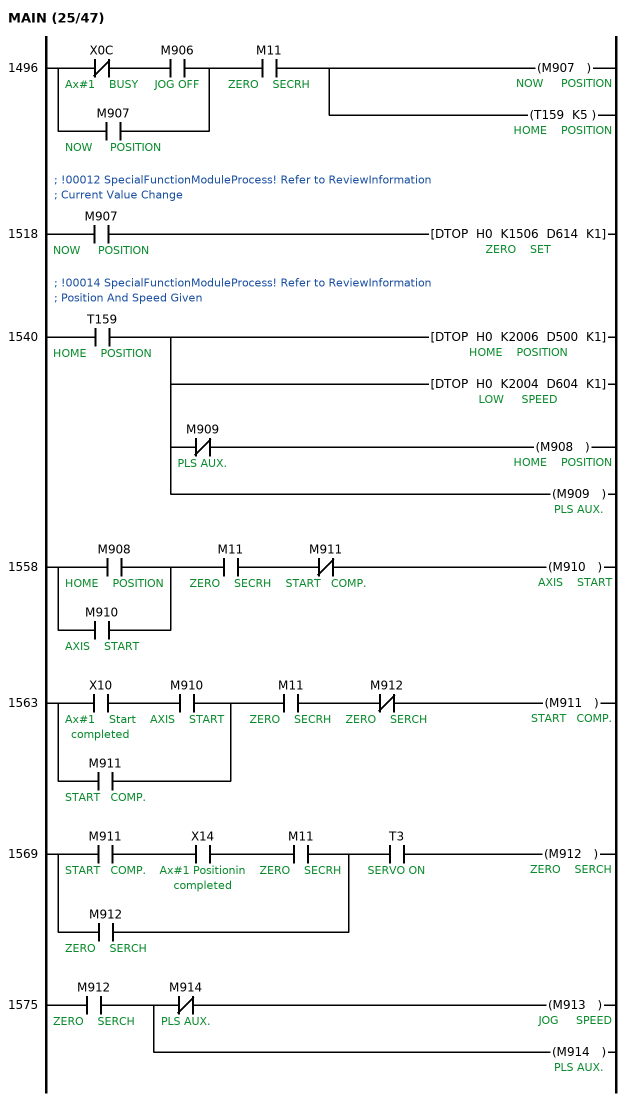
[picture p24: ladder of MAIN, rungs at steps 1496 to 1575]
1496  LDI     X0C  ; Ax#1    BUSY
      AND     M906  ; JOG OFF
      OR      M907  ; NOW     POSITION
      AND     M11  ; ZERO    SECRH
      OUT     M907  ; NOW     POSITION
      OUT     T159 K5  ; HOME    POSITION
; !00012 SpecialFunctionModuleProcess! Refer to ReviewInformation
; Current Value Change
1518  LD      M907  ; NOW     POSITION
      DTOP    H0 K1506 D614 K1
; !00014 SpecialFunctionModuleProcess! Refer to ReviewInformation
; Position And Speed Given
1540  LD      T159  ; HOME    POSITION
      DTOP    H0 K2006 D500 K1
      DTOP    H0 K2004 D604 K1
      MPS
      ANI     M909  ; PLS AUX.
      OUT     M908  ; HOME    POSITION
      MPP
      OUT     M909  ; PLS AUX.
1558  LD      M908  ; HOME    POSITION
      OR      M910  ; AXIS    START
      AND     M11  ; ZERO    SECRH
      ANI     M911  ; START   COMP.
      OUT     M910  ; AXIS    START
1563  LD      X10  ; Ax#1    Start   completed
      AND     M910  ; AXIS    START
      OR      M911  ; START   COMP.
      AND     M11  ; ZERO    SECRH
      ANI     M912  ; ZERO    SERCH
      OUT     M911  ; START   COMP.
1569  LD      M911  ; START   COMP.
      AND     X14  ; Ax#1 Positionin completed
      AND     M11  ; ZERO    SECRH
      OR      M912  ; ZERO    SERCH
      AND     T3  ; SERVO ON
      OUT     M912  ; ZERO    SERCH
1575  LD      M912  ; ZERO    SERCH
      MPS
      ANI     M914  ; PLS AUX.
      OUT     M913  ; JOG     SPEED
      MPP
      OUT     M914  ; PLS AUX.
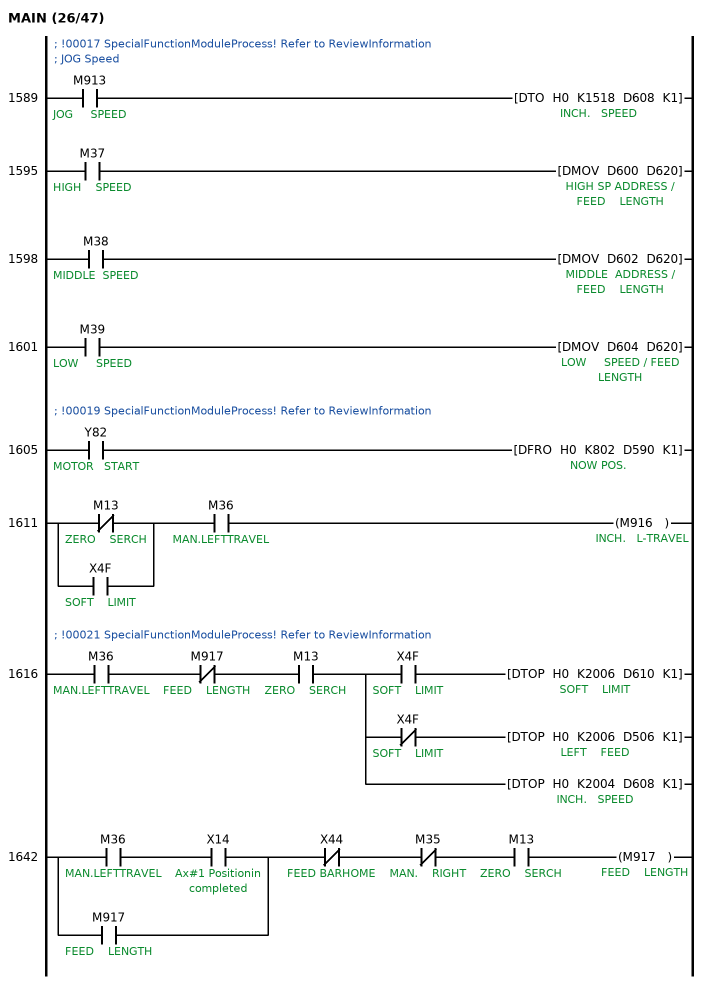
; !00017 SpecialFunctionModuleProcess! Refer to ReviewInformation
; JOG Speed
1589  LD      M913  ; JOG     SPEED
      DTO     H0 K1518 D608 K1
1595  LD      M37  ; HIGH    SPEED
      DMOV    D600 D620  ; FEED    LENGTH
1598  LD      M38  ; MIDDLE  SPEED
      DMOV    D602 D620
1601  LD      M39  ; LOW     SPEED
      DMOV    D604 D620
; !00019 SpecialFunctionModuleProcess! Refer to ReviewInformation
1605  LD      Y82  ; MOTOR   START
      DFRO    H0 K802 D590 K1
1611  LDI     M13  ; ZERO    SERCH
      OR      X4F  ; SOFT    LIMIT
      AND     M36  ; MAN.LEFTTRAVEL
      OUT     M916  ; INCH.   L-TRAVEL
; !00021 SpecialFunctionModuleProcess! Refer to ReviewInformation
1616  LD      M36  ; MAN.LEFTTRAVEL
      ANI     M917  ; FEED    LENGTH
      AND     M13  ; ZERO    SERCH
      MPS
      AND     X4F  ; SOFT    LIMIT
      DTOP    H0 K2006 D610 K1
      MRD
      ANI     X4F  ; SOFT    LIMIT
      DTOP    H0 K2006 D506 K1  ; LEFT    FEED
      MPP
      DTOP    H0 K2004 D608 K1
1642  LD      M36  ; MAN.LEFTTRAVEL
      AND     X14  ; Ax#1 Positionin completed
      OR      M917  ; FEED    LENGTH
      ANI     X44  ; FEED BARHOME
      ANI     M35  ; MAN.    RIGHT
      AND     M13  ; ZERO    SERCH
      OUT     M917  ; FEED    LENGTH
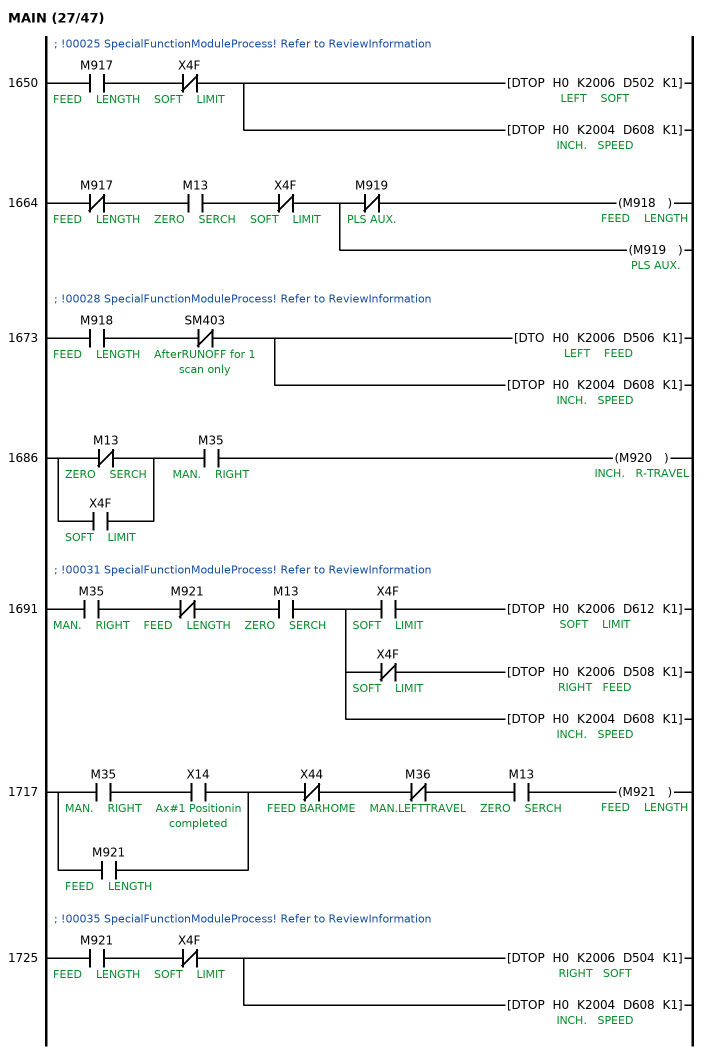
; !00025 SpecialFunctionModuleProcess! Refer to ReviewInformation
1650  LD      M917  ; FEED    LENGTH
      ANI     X4F  ; SOFT    LIMIT
      DTOP    H0 K2006 D502 K1
      DTOP    H0 K2004 D608 K1
1664  LDI     M917  ; FEED    LENGTH
      AND     M13  ; ZERO    SERCH
      ANI     X4F  ; SOFT    LIMIT
      MPS
      ANI     M919  ; PLS AUX.
      OUT     M918  ; FEED    LENGTH
      MPP
      OUT     M919  ; PLS AUX.
; !00028 SpecialFunctionModuleProcess! Refer to ReviewInformation
1673  LD      M918  ; FEED    LENGTH
      ANI     SM403  ; AfterRUNOFF for 1  scan only
      DTO     H0 K2006 D506 K1
      DTOP    H0 K2004 D608 K1
1686  LDI     M13  ; ZERO    SERCH
      OR      X4F  ; SOFT    LIMIT
      AND     M35  ; MAN.    RIGHT
      OUT     M920  ; INCH.   R-TRAVEL
; !00031 SpecialFunctionModuleProcess! Refer to ReviewInformation
1691  LD      M35  ; MAN.    RIGHT
      ANI     M921  ; FEED    LENGTH
      AND     M13  ; ZERO    SERCH
      MPS
      AND     X4F  ; SOFT    LIMIT
      DTOP    H0 K2006 D612 K1
      MRD
      ANI     X4F  ; SOFT    LIMIT
      DTOP    H0 K2006 D508 K1  ; RIGHT   FEED
      MPP
      DTOP    H0 K2004 D608 K1
1717  LD      M35  ; MAN.    RIGHT
      AND     X14  ; Ax#1 Positionin completed
      OR      M921  ; FEED    LENGTH
      ANI     X44  ; FEED BARHOME
      ANI     M36  ; MAN.LEFTTRAVEL
      AND     M13  ; ZERO    SERCH
      OUT     M921  ; FEED    LENGTH
; !00035 SpecialFunctionModuleProcess! Refer to ReviewInformation
1725  LD      M921  ; FEED    LENGTH
      ANI     X4F  ; SOFT    LIMIT
      DTOP    H0 K2006 D504 K1
      DTOP    H0 K2004 D608 K1
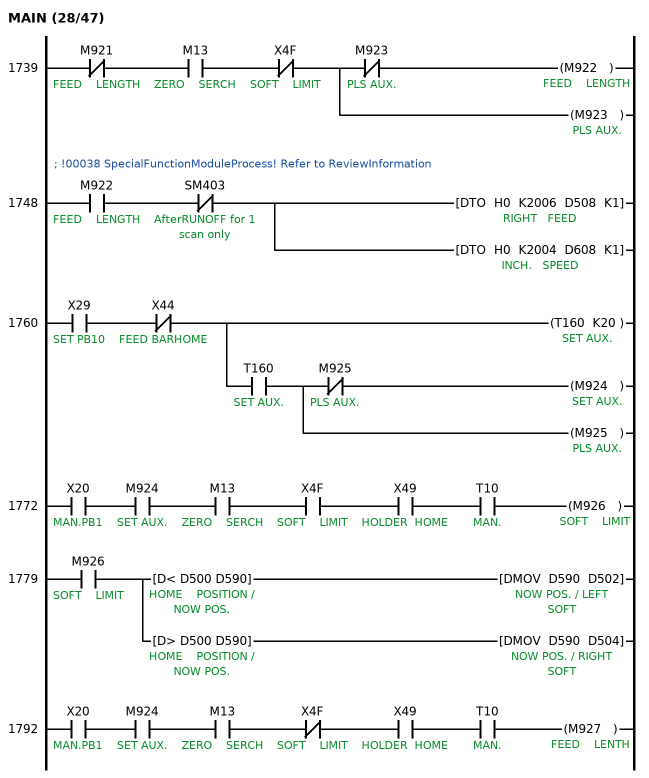
1739  LDI     M921  ; FEED    LENGTH
      AND     M13  ; ZERO    SERCH
      ANI     X4F  ; SOFT    LIMIT
      MPS
      ANI     M923  ; PLS AUX.
      OUT     M922  ; FEED    LENGTH
      MPP
      OUT     M923  ; PLS AUX.
; !00038 SpecialFunctionModuleProcess! Refer to ReviewInformation
1748  LD      M922  ; FEED    LENGTH
      ANI     SM403  ; AfterRUNOFF for 1  scan only
      DTO     H0 K2006 D508 K1
      DTO     H0 K2004 D608 K1
1760  LD      X29  ; SET PB10
      ANI     X44  ; FEED BARHOME
      OUT     T160 K20  ; SET AUX.
      AND     T160  ; SET AUX.
      MPS
      ANI     M925  ; PLS AUX.
      OUT     M924  ; SET AUX.
      MPP
      OUT     M925  ; PLS AUX.
1772  LD      X20  ; MAN.PB1
      AND     M924  ; SET AUX.
      AND     M13  ; ZERO    SERCH
      AND     X4F  ; SOFT    LIMIT
      AND     X49  ; HOLDER  HOME
      AND     T10  ; MAN.
      OUT     M926  ; SOFT    LIMIT
1779  LD      M926  ; SOFT    LIMIT
      MPS
      ANDD<   D500 D590  ; HOME    POSITION / NOW POS.
      DMOV    D590 D502
      MPP
      ANDD>   D500 D590  ; HOME    POSITION / NOW POS.
      DMOV    D590 D504
1792  LD      X20  ; MAN.PB1
      AND     M924  ; SET AUX.
      AND     M13  ; ZERO    SERCH
      ANI     X4F  ; SOFT    LIMIT
      AND     X49  ; HOLDER  HOME
      AND     T10  ; MAN.
      OUT     M927  ; FEED    LENTH
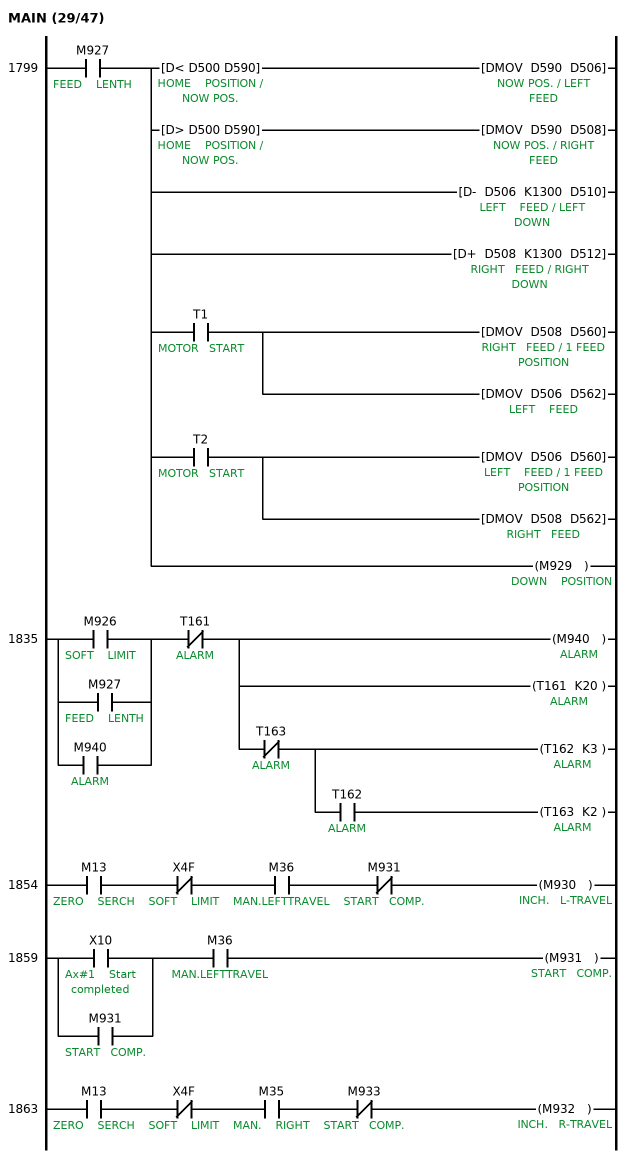
1799  LD      M927  ; FEED    LENTH
      MPS
      ANDD<   D500 D590  ; HOME    POSITION / NOW POS.
      DMOV    D590 D506
      MRD
      ANDD>   D500 D590  ; HOME    POSITION / NOW POS.
      DMOV    D590 D508
      MPP
      D-      D506 K1300 D510  ; LEFT    DOWN
      D+      D508 K1300 D512  ; RIGHT   DOWN
      MPS
      AND     T1  ; MOTOR   START
      DMOV    D508 D560  ; 1 FEED  POSITION
      DMOV    D506 D562
      MRD
      AND     T2  ; MOTOR   START
      DMOV    D506 D560
      DMOV    D508 D562
      MPP
      OUT     M929  ; DOWN    POSITION
1835  LD      M926  ; SOFT    LIMIT
      OR      M927  ; FEED    LENTH
      OR      M940  ; ALARM
      ANI     T161  ; ALARM
      OUT     M940  ; ALARM
      OUT     T161 K20  ; ALARM
      ANI     T163  ; ALARM
      OUT     T162 K3  ; ALARM
      AND     T162  ; ALARM
      OUT     T163 K2  ; ALARM
1854  LD      M13  ; ZERO    SERCH
      ANI     X4F  ; SOFT    LIMIT
      AND     M36  ; MAN.LEFTTRAVEL
      ANI     M931  ; START   COMP.
      OUT     M930  ; INCH.   L-TRAVEL
1859  LD      X10  ; Ax#1    Start   completed
      OR      M931  ; START   COMP.
      AND     M36  ; MAN.LEFTTRAVEL
      OUT     M931  ; START   COMP.
1863  LD      M13  ; ZERO    SERCH
      ANI     X4F  ; SOFT    LIMIT
      AND     M35  ; MAN.    RIGHT
      ANI     M933  ; START   COMP.
      OUT     M932  ; INCH.   R-TRAVEL
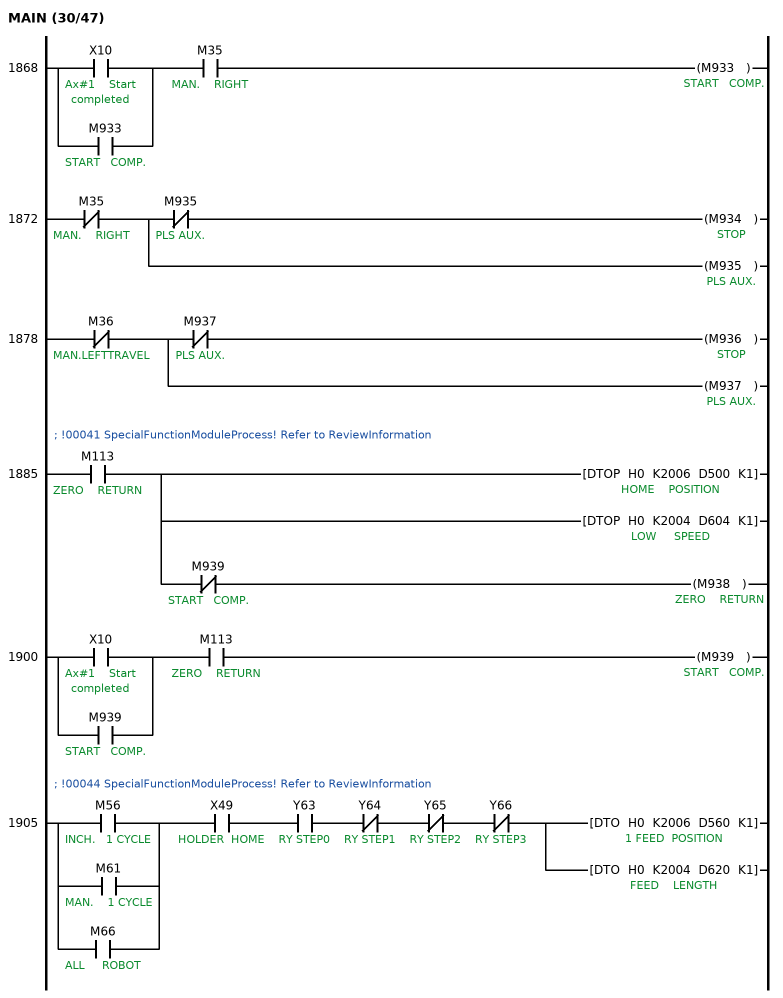
1868  LD      X10  ; Ax#1    Start   completed
      OR      M933  ; START   COMP.
      AND     M35  ; MAN.    RIGHT
      OUT     M933  ; START   COMP.
1872  LDI     M35  ; MAN.    RIGHT
      MPS
      ANI     M935  ; PLS AUX.
      OUT     M934  ; STOP
      MPP
      OUT     M935  ; PLS AUX.
1878  LDI     M36  ; MAN.LEFTTRAVEL
      MPS
      ANI     M937  ; PLS AUX.
      OUT     M936  ; STOP
      MPP
      OUT     M937  ; PLS AUX.
; !00041 SpecialFunctionModuleProcess! Refer to ReviewInformation
1885  LD      M113  ; ZERO    RETURN
      DTOP    H0 K2006 D500 K1
      DTOP    H0 K2004 D604 K1
      ANI     M939  ; START   COMP.
      OUT     M938  ; ZERO    RETURN
1900  LD      X10  ; Ax#1    Start   completed
      OR      M939  ; START   COMP.
      AND     M113  ; ZERO    RETURN
      OUT     M939  ; START   COMP.
; !00044 SpecialFunctionModuleProcess! Refer to ReviewInformation
1905  LD      M56  ; INCH.   1 CYCLE
      OR      M61  ; MAN.    1 CYCLE
      OR      M66  ; ALL     ROBOT
      AND     X49  ; HOLDER  HOME
      AND     Y63  ; RY STEP0
      ANI     Y64  ; RY STEP1
      ANI     Y65  ; RY STEP2
      ANI     Y66  ; RY STEP3
      DTO     H0 K2006 D560 K1
      DTO     H0 K2004 D620 K1
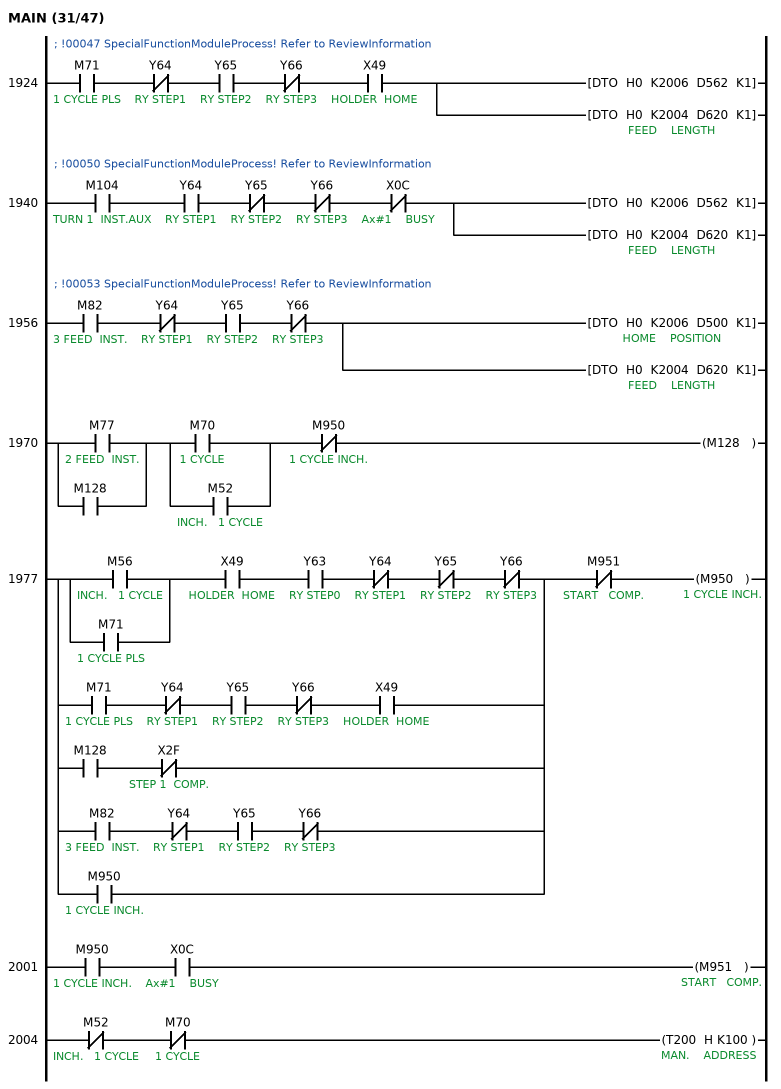
; !00047 SpecialFunctionModuleProcess! Refer to ReviewInformation
1924  LD      M71  ; 1 CYCLE PLS
      ANI     Y64  ; RY STEP1
      AND     Y65  ; RY STEP2
      ANI     Y66  ; RY STEP3
      AND     X49  ; HOLDER  HOME
      DTO     H0 K2006 D562 K1
      DTO     H0 K2004 D620 K1
; !00050 SpecialFunctionModuleProcess! Refer to ReviewInformation
1940  LD      M104  ; TURN 1  INST.AUX
      AND     Y64  ; RY STEP1
      ANI     Y65  ; RY STEP2
      ANI     Y66  ; RY STEP3
      ANI     X0C  ; Ax#1    BUSY
      DTO     H0 K2006 D562 K1
      DTO     H0 K2004 D620 K1
; !00053 SpecialFunctionModuleProcess! Refer to ReviewInformation
1956  LD      M82  ; 3 FEED  INST.
      ANI     Y64  ; RY STEP1
      AND     Y65  ; RY STEP2
      ANI     Y66  ; RY STEP3
      DTO     H0 K2006 D500 K1
      DTO     H0 K2004 D620 K1
1970  LD      M77  ; 2 FEED  INST.
      OR      M128
      LD      M70  ; 1 CYCLE
      OR      M52  ; INCH.   1 CYCLE
      ANB
      ANI     M950  ; 1 CYCLE INCH.
      OUT     M128
1977  LD      M56  ; INCH.   1 CYCLE
      OR      M71  ; 1 CYCLE PLS
      AND     X49  ; HOLDER  HOME
      AND     Y63  ; RY STEP0
      ANI     Y64  ; RY STEP1
      ANI     Y65  ; RY STEP2
      ANI     Y66  ; RY STEP3
      LD      M71  ; 1 CYCLE PLS
      ANI     Y64  ; RY STEP1
      AND     Y65  ; RY STEP2
      ANI     Y66  ; RY STEP3
      AND     X49  ; HOLDER  HOME
      ORB
      LD      M128
      ANI     X2F  ; STEP 1  COMP.
      ORB
      LD      M82  ; 3 FEED  INST.
      ANI     Y64  ; RY STEP1
      AND     Y65  ; RY STEP2
      ANI     Y66  ; RY STEP3
      ORB
      OR      M950  ; 1 CYCLE INCH.
      ANI     M951  ; START   COMP.
      OUT     M950  ; 1 CYCLE INCH.
2001  LD      M950  ; 1 CYCLE INCH.
      AND     X0C  ; Ax#1    BUSY
      OUT     M951  ; START   COMP.
2004  LDI     M52  ; INCH.   1 CYCLE
      ANI     M70  ; 1 CYCLE
      OUTH    T200 K100  ; MAN.    ADDRESS
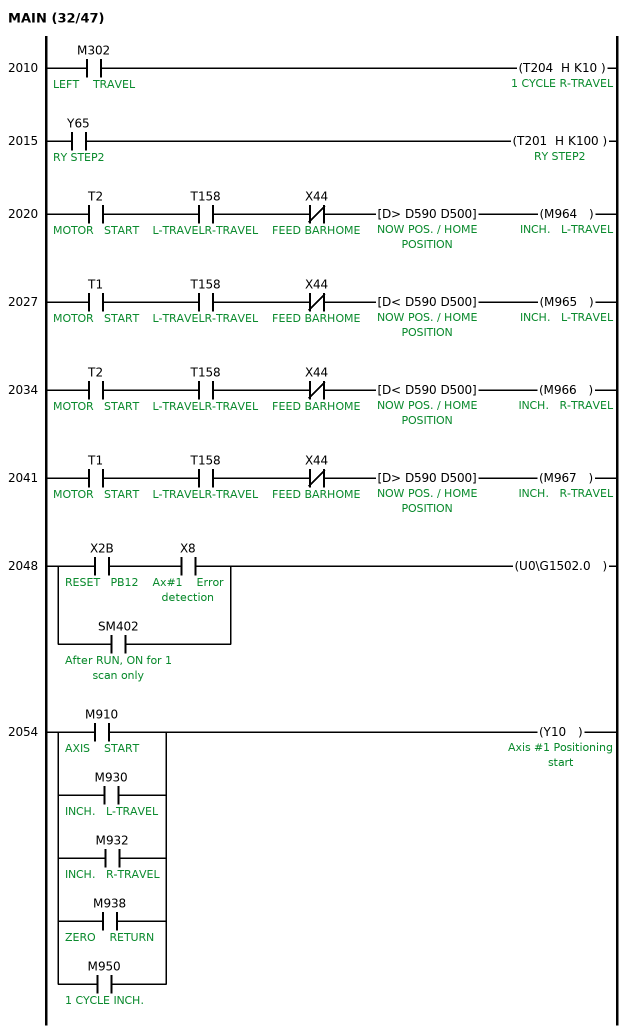
2010  LD      M302  ; LEFT    TRAVEL
      OUTH    T204 K10  ; 1 CYCLE R-TRAVEL
2015  LD      Y65  ; RY STEP2
      OUTH    T201 K100  ; RY STEP2
2020  LD      T2  ; MOTOR   START
      AND     T158  ; L-TRAVELR-TRAVEL
      ANI     X44  ; FEED BARHOME
      ANDD>   D590 D500  ; NOW POS. / HOME    POSITION
      OUT     M964  ; INCH.   L-TRAVEL
2027  LD      T1  ; MOTOR   START
      AND     T158  ; L-TRAVELR-TRAVEL
      ANI     X44  ; FEED BARHOME
      ANDD<   D590 D500  ; NOW POS. / HOME    POSITION
      OUT     M965  ; INCH.   L-TRAVEL
2034  LD      T2  ; MOTOR   START
      AND     T158  ; L-TRAVELR-TRAVEL
      ANI     X44  ; FEED BARHOME
      ANDD<   D590 D500  ; NOW POS. / HOME    POSITION
      OUT     M966  ; INCH.   R-TRAVEL
2041  LD      T1  ; MOTOR   START
      AND     T158  ; L-TRAVELR-TRAVEL
      ANI     X44  ; FEED BARHOME
      ANDD>   D590 D500  ; NOW POS. / HOME    POSITION
      OUT     M967  ; INCH.   R-TRAVEL
2048  LD      X2B  ; RESET   PB12
      AND     X8  ; Ax#1    Error   detection
      OR      SM402  ; After RUN, ON for 1 scan only
      OUT     U0\G1502.0
2054  LD      M910  ; AXIS    START
      OR      M930  ; INCH.   L-TRAVEL
      OR      M932  ; INCH.   R-TRAVEL
      OR      M938  ; ZERO    RETURN
      OR      M950  ; 1 CYCLE INCH.
      OUT     Y10  ; Axis #1 Positioning start
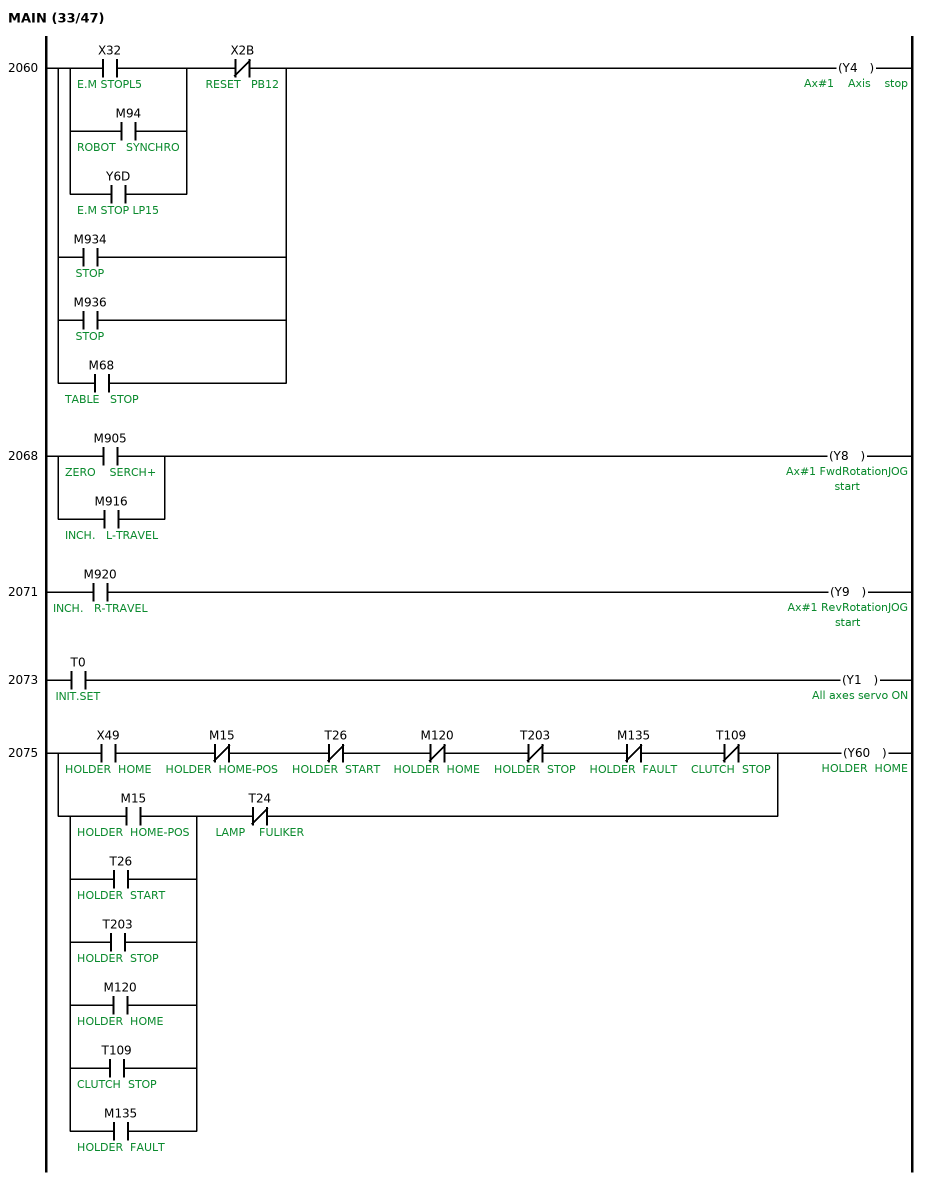
2060  LD      X32  ; E.M STOPL5
      OR      M94  ; ROBOT   SYNCHRO
      OR      Y6D  ; E.M STOP LP15
      ANI     X2B  ; RESET   PB12
      OR      M934  ; STOP
      OR      M936  ; STOP
      OR      M68  ; TABLE   STOP
      OUT     Y4  ; Ax#1    Axis    stop
2068  LD      M905  ; ZERO    SERCH+
      OR      M916  ; INCH.   L-TRAVEL
      OUT     Y8  ; Ax#1 FwdRotationJOG     start
2071  LD      M920  ; INCH.   R-TRAVEL
      OUT     Y9  ; Ax#1 RevRotationJOG     start
2073  LD      T0  ; INIT.SET
      OUT     Y1  ; All axes servo ON
2075  LD      X49  ; HOLDER  HOME
      ANI     M15  ; HOLDER  HOME-POS
      ANI     T26  ; HOLDER  START
      ANI     M120  ; HOLDER  HOME
      ANI     T203  ; HOLDER  STOP
      ANI     M135  ; HOLDER  FAULT
      ANI     T109  ; CLUTCH  STOP
      LD      M15  ; HOLDER  HOME-POS
      OR      T26  ; HOLDER  START
      OR      T203  ; HOLDER  STOP
      OR      M120  ; HOLDER  HOME
      OR      T109  ; CLUTCH  STOP
      OR      M135  ; HOLDER  FAULT
      ANI     T24  ; LAMP    FULIKER
      ORB
      OUT     Y60  ; HOLDER  HOME
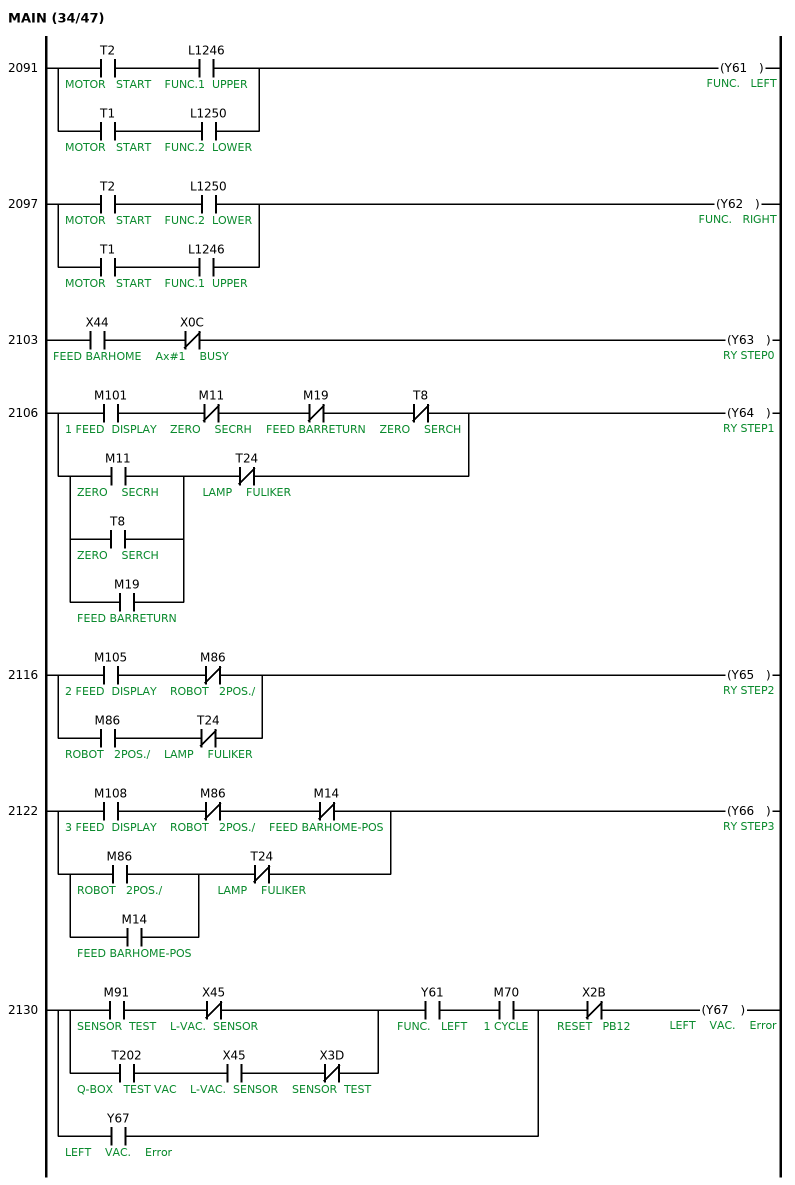
2091  LD      T2  ; MOTOR   START
      AND     L1246  ; FUNC.1  UPPER
      LD      T1  ; MOTOR   START
      AND     L1250  ; FUNC.2  LOWER
      ORB
      OUT     Y61  ; FUNC.   LEFT
2097  LD      T2  ; MOTOR   START
      AND     L1250  ; FUNC.2  LOWER
      LD      T1  ; MOTOR   START
      AND     L1246  ; FUNC.1  UPPER
      ORB
      OUT     Y62  ; FUNC.   RIGHT
2103  LD      X44  ; FEED BARHOME
      ANI     X0C  ; Ax#1    BUSY
      OUT     Y63  ; RY STEP0
2106  LD      M101  ; 1 FEED  DISPLAY
      ANI     M11  ; ZERO    SECRH
      ANI     M19  ; FEED BARRETURN
      ANI     T8  ; ZERO    SERCH
      LD      M11  ; ZERO    SECRH
      OR      T8  ; ZERO    SERCH
      OR      M19  ; FEED BARRETURN
      ANI     T24  ; LAMP    FULIKER
      ORB
      OUT     Y64  ; RY STEP1
2116  LD      M105  ; 2 FEED  DISPLAY
      ANI     M86  ; ROBOT   2POS./
      LD      M86  ; ROBOT   2POS./
      ANI     T24  ; LAMP    FULIKER
      ORB
      OUT     Y65  ; RY STEP2
2122  LD      M108  ; 3 FEED  DISPLAY
      ANI     M86  ; ROBOT   2POS./
      ANI     M14  ; FEED BARHOME-POS
      LD      M86  ; ROBOT   2POS./
      OR      M14  ; FEED BARHOME-POS
      ANI     T24  ; LAMP    FULIKER
      ORB
      OUT     Y66  ; RY STEP3
2130  LD      M91  ; SENSOR  TEST
      ANI     X45  ; L-VAC.  SENSOR
      LD      T202  ; Q-BOX   TEST VAC
      AND     X45  ; L-VAC.  SENSOR
      ANI     X3D  ; SENSOR  TEST
      ORB
      AND     Y61  ; FUNC.   LEFT
      AND     M70  ; 1 CYCLE
      OR      Y67  ; LEFT    VAC.    Error
      ANI     X2B  ; RESET   PB12
      OUT     Y67  ; LEFT    VAC.    Error
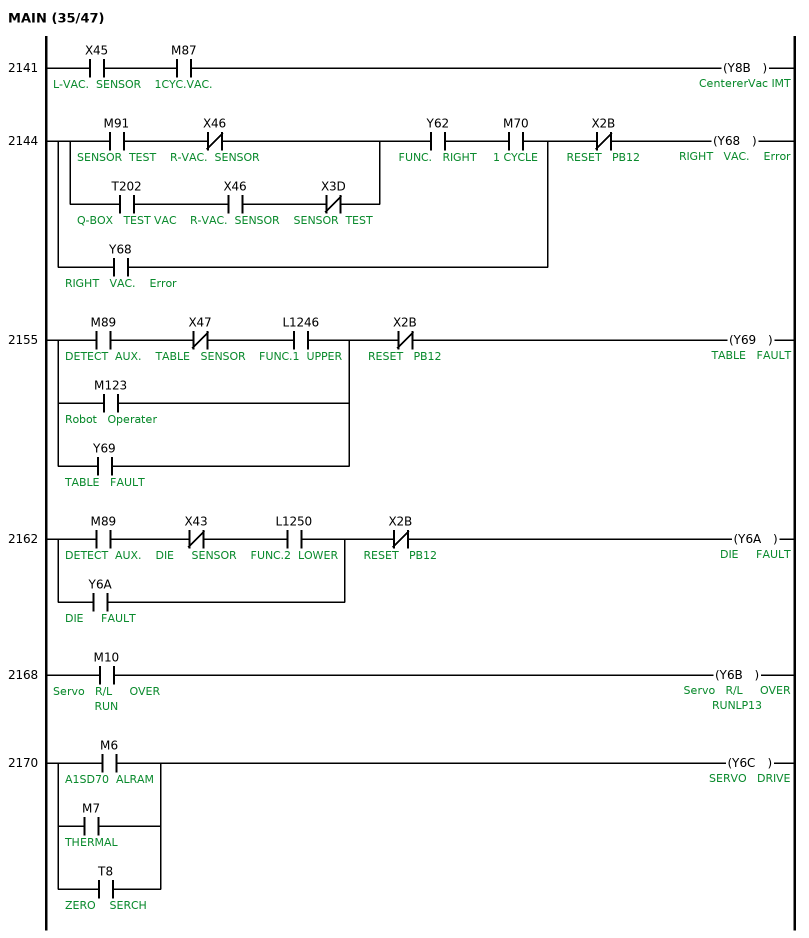
2141  LD      X45  ; L-VAC.  SENSOR
      AND     M87  ; 1CYC.VAC.
      OUT     Y8B  ; CentererVac IMT
2144  LD      M91  ; SENSOR  TEST
      ANI     X46  ; R-VAC.  SENSOR
      LD      T202  ; Q-BOX   TEST VAC
      AND     X46  ; R-VAC.  SENSOR
      ANI     X3D  ; SENSOR  TEST
      ORB
      AND     Y62  ; FUNC.   RIGHT
      AND     M70  ; 1 CYCLE
      OR      Y68  ; RIGHT   VAC.    Error
      ANI     X2B  ; RESET   PB12
      OUT     Y68  ; RIGHT   VAC.    Error
2155  LD      M89  ; DETECT  AUX.
      ANI     X47  ; TABLE   SENSOR
      AND     L1246  ; FUNC.1  UPPER
      OR      M123  ; Robot   Operater
      OR      Y69  ; TABLE   FAULT
      ANI     X2B  ; RESET   PB12
      OUT     Y69  ; TABLE   FAULT
2162  LD      M89  ; DETECT  AUX.
      ANI     X43  ; DIE     SENSOR
      AND     L1250  ; FUNC.2  LOWER
      OR      Y6A  ; DIE     FAULT
      ANI     X2B  ; RESET   PB12
      OUT     Y6A  ; DIE     FAULT
2168  LD      M10  ; Servo   R/L     OVER RUN
      OUT     Y6B  ; Servo   R/L     OVER RUNLP13
2170  LD      M6  ; A1SD70  ALRAM
      OR      M7  ; THERMAL
      OR      T8  ; ZERO    SERCH
      OUT     Y6C  ; SERVO   DRIVE
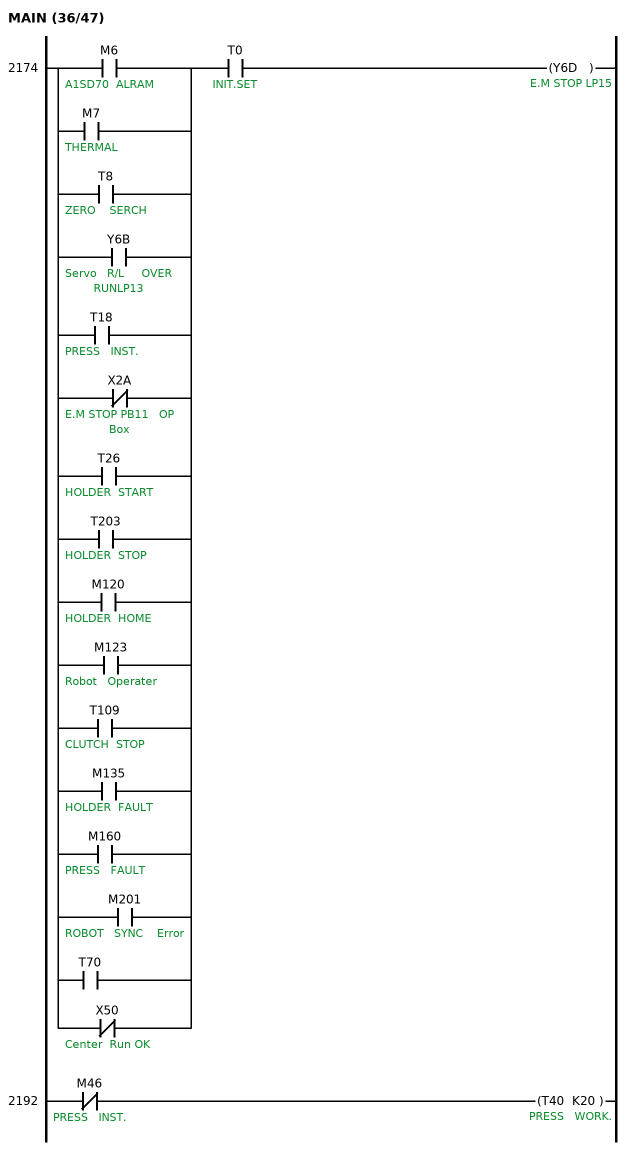
2174  LD      M6  ; A1SD70  ALRAM
      OR      M7  ; THERMAL
      OR      T8  ; ZERO    SERCH
      OR      Y6B  ; Servo   R/L     OVER RUNLP13
      OR      T18  ; PRESS   INST.
      ORI     X2A  ; E.M STOP PB11   OP Box
      OR      T26  ; HOLDER  START
      OR      T203  ; HOLDER  STOP
      OR      M120  ; HOLDER  HOME
      OR      M123  ; Robot   Operater
      OR      T109  ; CLUTCH  STOP
      OR      M135  ; HOLDER  FAULT
      OR      M160  ; PRESS   FAULT
      OR      M201  ; ROBOT   SYNC    Error
      OR      T70
      ORI     X50  ; Center  Run OK
      AND     T0  ; INIT.SET
      OUT     Y6D  ; E.M STOP LP15
2192  LDI     M46  ; PRESS   INST.
      OUT     T40 K20  ; PRESS   WORK.
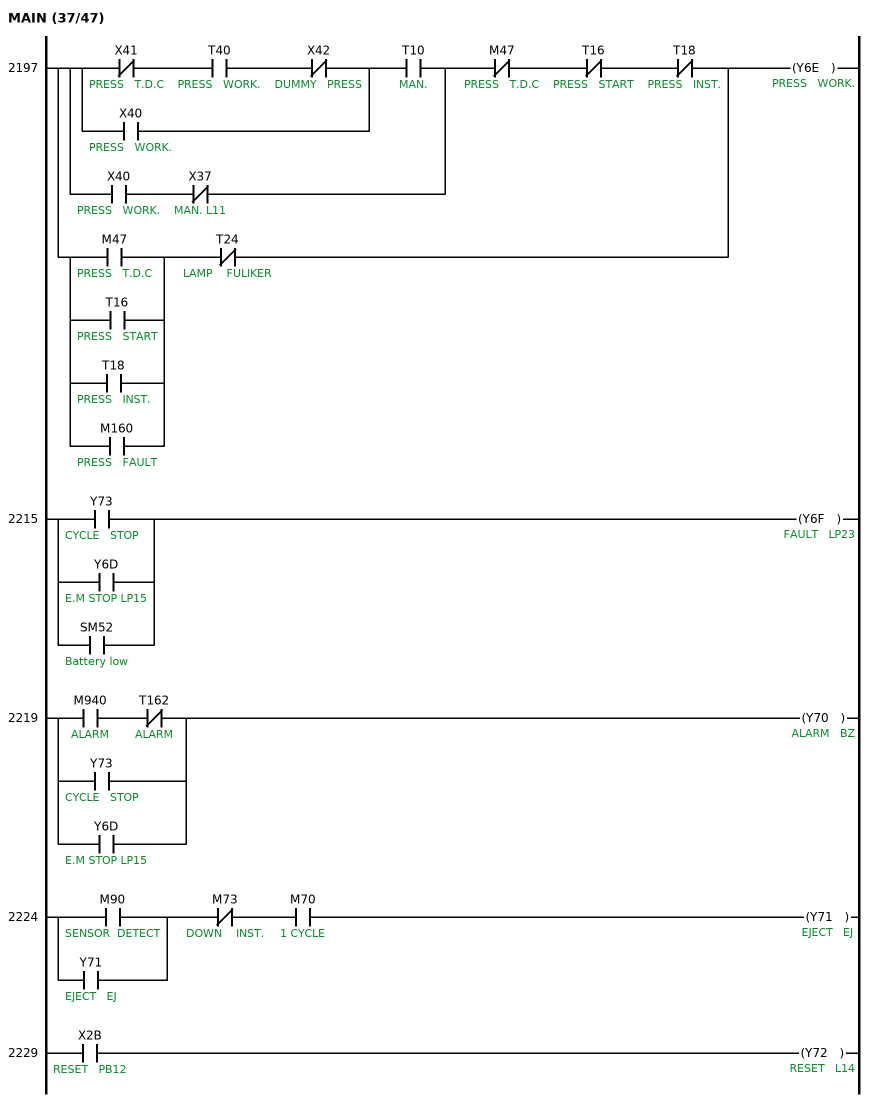
2197  LDI     X41  ; PRESS   T.D.C
      AND     T40  ; PRESS   WORK.
      ANI     X42  ; DUMMY   PRESS
      OR      X40  ; PRESS   WORK.
      AND     T10  ; MAN.
      LD      X40  ; PRESS   WORK.
      ANI     X37  ; MAN. L11
      ORB
      ANI     M47  ; PRESS   T.D.C
      ANI     T16  ; PRESS   START
      ANI     T18  ; PRESS   INST.
      LD      M47  ; PRESS   T.D.C
      OR      T16  ; PRESS   START
      OR      T18  ; PRESS   INST.
      OR      M160  ; PRESS   FAULT
      ANI     T24  ; LAMP    FULIKER
      ORB
      OUT     Y6E  ; PRESS   WORK.
2215  LD      Y73  ; CYCLE   STOP
      OR      Y6D  ; E.M STOP LP15
      OR      SM52  ; Battery low
      OUT     Y6F  ; FAULT   LP23
2219  LD      M940  ; ALARM
      ANI     T162  ; ALARM
      OR      Y73  ; CYCLE   STOP
      OR      Y6D  ; E.M STOP LP15
      OUT     Y70  ; ALARM   BZ
2224  LD      M90  ; SENSOR  DETECT
      OR      Y71  ; EJECT   EJ
      ANI     M73  ; DOWN    INST.
      AND     M70  ; 1 CYCLE
      OUT     Y71  ; EJECT   EJ
2229  LD      X2B  ; RESET   PB12
      OUT     Y72  ; RESET   L14
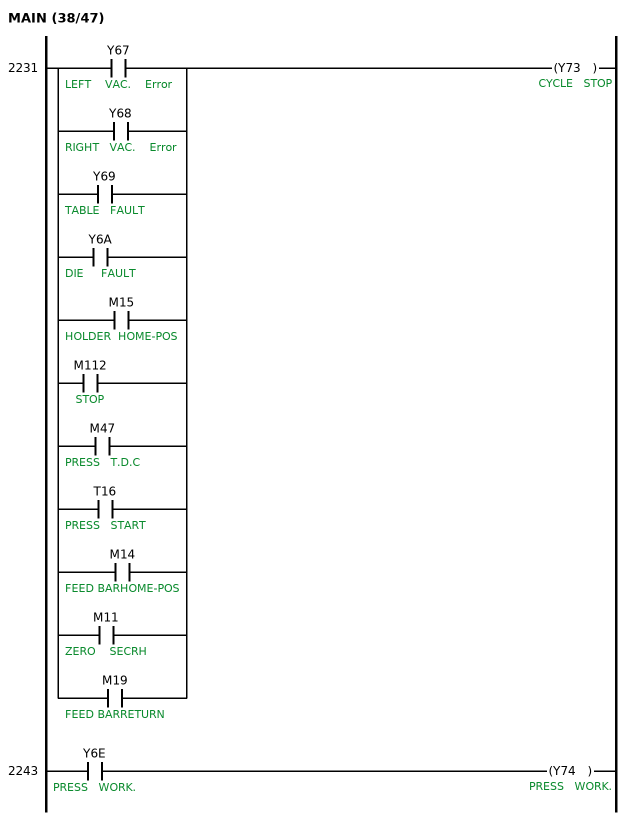
2231  LD      Y67  ; LEFT    VAC.    Error
      OR      Y68  ; RIGHT   VAC.    Error
      OR      Y69  ; TABLE   FAULT
      OR      Y6A  ; DIE     FAULT
      OR      M15  ; HOLDER  HOME-POS
      OR      M112  ; STOP
      OR      M47  ; PRESS   T.D.C
      OR      T16  ; PRESS   START
      OR      M14  ; FEED BARHOME-POS
      OR      M11  ; ZERO    SECRH
      OR      M19  ; FEED BARRETURN
      OUT     Y73  ; CYCLE   STOP
2243  LD      Y6E  ; PRESS   WORK.
      OUT     Y74  ; PRESS   WORK.
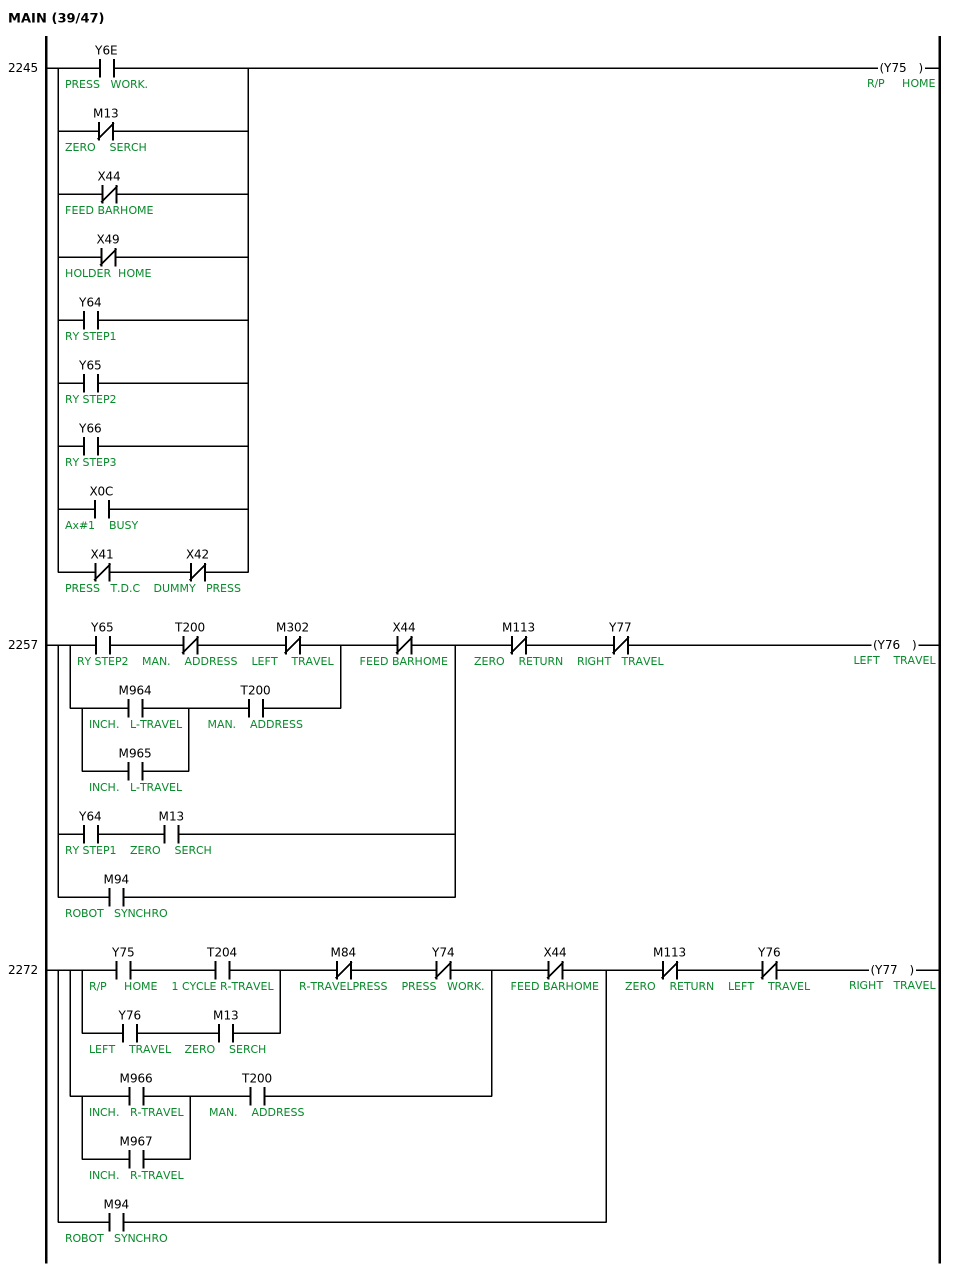
2245  LD      Y6E  ; PRESS   WORK.
      ORI     M13  ; ZERO    SERCH
      ORI     X44  ; FEED BARHOME
      ORI     X49  ; HOLDER  HOME
      OR      Y64  ; RY STEP1
      OR      Y65  ; RY STEP2
      OR      Y66  ; RY STEP3
      OR      X0C  ; Ax#1    BUSY
      LDI     X41  ; PRESS   T.D.C
      ANI     X42  ; DUMMY   PRESS
      ORB
      OUT     Y75  ; R/P     HOME
2257  LD      Y65  ; RY STEP2
      ANI     T200  ; MAN.    ADDRESS
      ANI     M302  ; LEFT    TRAVEL
      LD      M964  ; INCH.   L-TRAVEL
      OR      M965  ; INCH.   L-TRAVEL
      AND     T200  ; MAN.    ADDRESS
      ORB
      ANI     X44  ; FEED BARHOME
      LD      Y64  ; RY STEP1
      AND     M13  ; ZERO    SERCH
      ORB
      OR      M94  ; ROBOT   SYNCHRO
      ANI     M113  ; ZERO    RETURN
      ANI     Y77  ; RIGHT   TRAVEL
      OUT     Y76  ; LEFT    TRAVEL
2272  LD      Y75  ; R/P     HOME
      AND     T204  ; 1 CYCLE R-TRAVEL
      LD      Y76  ; LEFT    TRAVEL
      AND     M13  ; ZERO    SERCH
      ORB
      ANI     M84  ; R-TRAVELPRESS
      ANI     Y74  ; PRESS   WORK.
      LD      M966  ; INCH.   R-TRAVEL
      OR      M967  ; INCH.   R-TRAVEL
      AND     T200  ; MAN.    ADDRESS
      ORB
      ANI     X44  ; FEED BARHOME
      OR      M94  ; ROBOT   SYNCHRO
      ANI     M113  ; ZERO    RETURN
      ANI     Y76  ; LEFT    TRAVEL
      OUT     Y77  ; RIGHT   TRAVEL
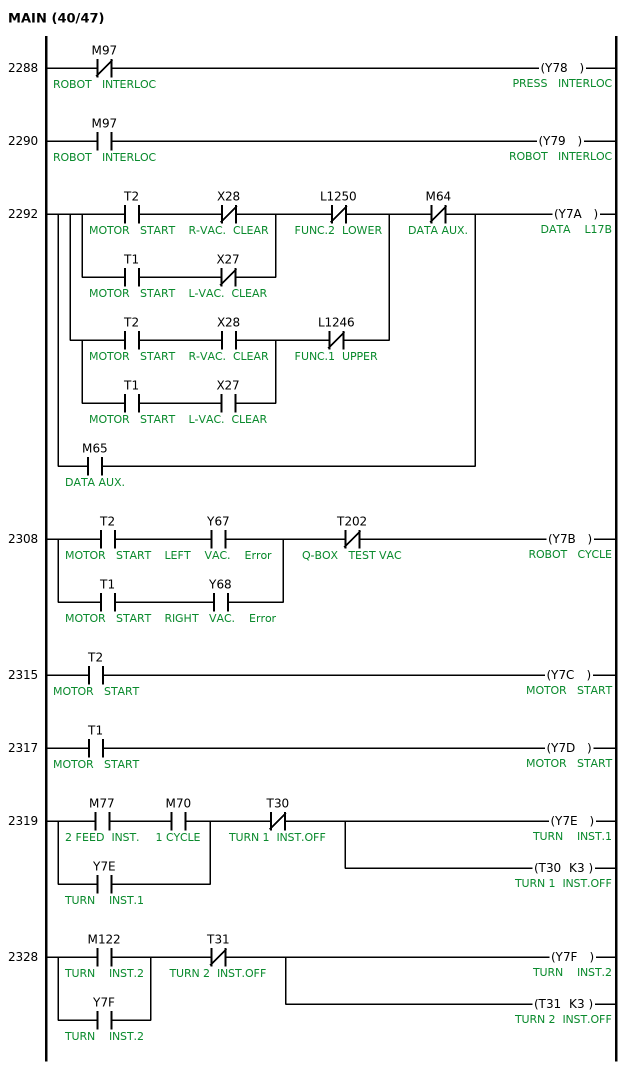
2288  LDI     M97  ; ROBOT   INTERLOC
      OUT     Y78  ; PRESS   INTERLOC
2290  LD      M97  ; ROBOT   INTERLOC
      OUT     Y79  ; ROBOT   INTERLOC
2292  LD      T2  ; MOTOR   START
      ANI     X28  ; R-VAC.  CLEAR
      LD      T1  ; MOTOR   START
      ANI     X27  ; L-VAC.  CLEAR
      ORB
      ANI     L1250  ; FUNC.2  LOWER
      LD      T2  ; MOTOR   START
      AND     X28  ; R-VAC.  CLEAR
      LD      T1  ; MOTOR   START
      AND     X27  ; L-VAC.  CLEAR
      ORB
      ANI     L1246  ; FUNC.1  UPPER
      ORB
      ANI     M64  ; DATA AUX.
      OR      M65  ; DATA AUX.
      OUT     Y7A  ; DATA    L17B
2308  LD      T2  ; MOTOR   START
      AND     Y67  ; LEFT    VAC.    Error
      LD      T1  ; MOTOR   START
      AND     Y68  ; RIGHT   VAC.    Error
      ORB
      ANI     T202  ; Q-BOX   TEST VAC
      OUT     Y7B  ; ROBOT   CYCLE
2315  LD      T2  ; MOTOR   START
      OUT     Y7C  ; MOTOR   START
2317  LD      T1  ; MOTOR   START
      OUT     Y7D  ; MOTOR   START
2319  LD      M77  ; 2 FEED  INST.
      AND     M70  ; 1 CYCLE
      OR      Y7E  ; TURN    INST.1
      ANI     T30  ; TURN 1  INST.OFF
      OUT     Y7E  ; TURN    INST.1
      OUT     T30 K3  ; TURN 1  INST.OFF
2328  LD      M122  ; TURN    INST.2
      OR      Y7F  ; TURN    INST.2
      ANI     T31  ; TURN 2  INST.OFF
      OUT     Y7F  ; TURN    INST.2
      OUT     T31 K3  ; TURN 2  INST.OFF
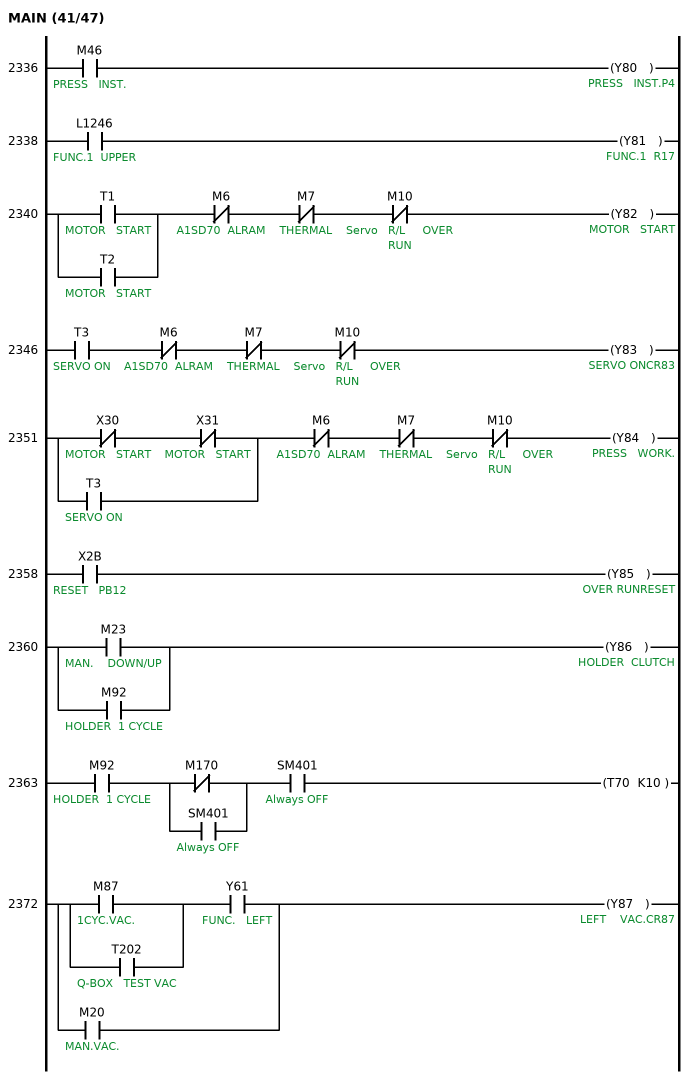
2336  LD      M46  ; PRESS   INST.
      OUT     Y80  ; PRESS   INST.P4
2338  LD      L1246  ; FUNC.1  UPPER
      OUT     Y81  ; FUNC.1  R17
2340  LD      T1  ; MOTOR   START
      OR      T2  ; MOTOR   START
      ANI     M6  ; A1SD70  ALRAM
      ANI     M7  ; THERMAL
      ANI     M10  ; Servo   R/L     OVER RUN
      OUT     Y82  ; MOTOR   START
2346  LD      T3  ; SERVO ON
      ANI     M6  ; A1SD70  ALRAM
      ANI     M7  ; THERMAL
      ANI     M10  ; Servo   R/L     OVER RUN
      OUT     Y83  ; SERVO ONCR83
2351  LDI     X30  ; MOTOR   START
      ANI     X31  ; MOTOR   START
      OR      T3  ; SERVO ON
      ANI     M6  ; A1SD70  ALRAM
      ANI     M7  ; THERMAL
      ANI     M10  ; Servo   R/L     OVER RUN
      OUT     Y84  ; PRESS   WORK.
2358  LD      X2B  ; RESET   PB12
      OUT     Y85  ; OVER RUNRESET
2360  LD      M23  ; MAN.    DOWN/UP
      OR      M92  ; HOLDER  1 CYCLE
      OUT     Y86  ; HOLDER  CLUTCH
2363  LD      M92  ; HOLDER  1 CYCLE
      LDI     M170
      OR      SM401  ; Always OFF
      ANB
      AND     SM401  ; Always OFF
      OUT     T70 K10
2372  LD      M87  ; 1CYC.VAC.
      OR      T202  ; Q-BOX   TEST VAC
      AND     Y61  ; FUNC.   LEFT
      OR      M20  ; MAN.VAC.
      OUT     Y87  ; LEFT    VAC.CR87
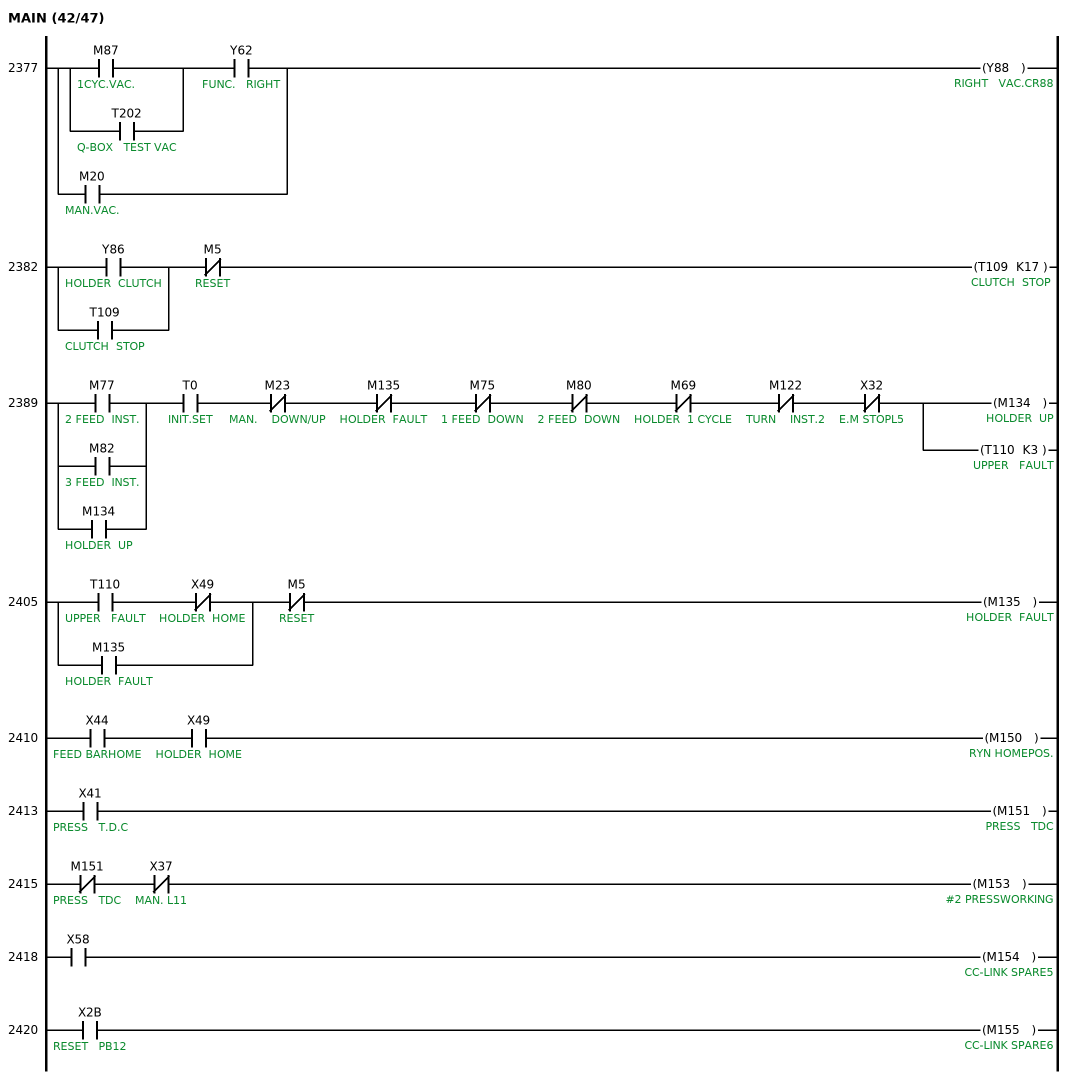
2377  LD      M87  ; 1CYC.VAC.
      OR      T202  ; Q-BOX   TEST VAC
      AND     Y62  ; FUNC.   RIGHT
      OR      M20  ; MAN.VAC.
      OUT     Y88  ; RIGHT   VAC.CR88
2382  LD      Y86  ; HOLDER  CLUTCH
      OR      T109  ; CLUTCH  STOP
      ANI     M5  ; RESET
      OUT     T109 K17  ; CLUTCH  STOP
2389  LD      M77  ; 2 FEED  INST.
      OR      M82  ; 3 FEED  INST.
      OR      M134  ; HOLDER  UP
      AND     T0  ; INIT.SET
      ANI     M23  ; MAN.    DOWN/UP
      ANI     M135  ; HOLDER  FAULT
      ANI     M75  ; 1 FEED  DOWN
      ANI     M80  ; 2 FEED  DOWN
      ANI     M69  ; HOLDER  1 CYCLE
      ANI     M122  ; TURN    INST.2
      ANI     X32  ; E.M STOPL5
      OUT     M134  ; HOLDER  UP
      OUT     T110 K3  ; UPPER   FAULT
2405  LD      T110  ; UPPER   FAULT
      ANI     X49  ; HOLDER  HOME
      OR      M135  ; HOLDER  FAULT
      ANI     M5  ; RESET
      OUT     M135  ; HOLDER  FAULT
2410  LD      X44  ; FEED BARHOME
      AND     X49  ; HOLDER  HOME
      OUT     M150  ; RYN HOMEPOS.
2413  LD      X41  ; PRESS   T.D.C
      OUT     M151  ; PRESS   TDC
2415  LDI     M151  ; PRESS   TDC
      ANI     X37  ; MAN. L11
      OUT     M153  ; #2 PRESSWORKING
2418  LD      X58
      OUT     M154  ; CC-LINK SPARE5
2420  LD      X2B  ; RESET   PB12
      OUT     M155  ; CC-LINK SPARE6
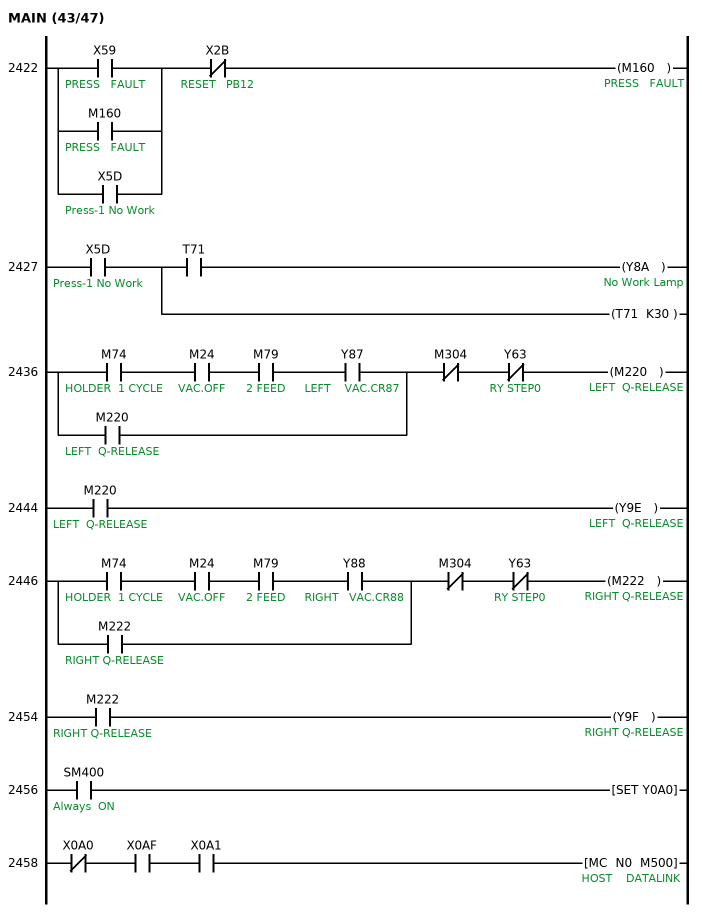
2422  LD      X59  ; PRESS   FAULT
      OR      M160  ; PRESS   FAULT
      OR      X5D  ; Press-1 No Work
      ANI     X2B  ; RESET   PB12
      OUT     M160  ; PRESS   FAULT
2427  LD      X5D  ; Press-1 No Work
      MPS
      AND     T71
      OUT     Y8A  ; No Work Lamp
      MPP
      OUT     T71 K30
2436  LD      M74  ; HOLDER  1 CYCLE
      AND     M24  ; VAC.OFF
      AND     M79  ; 2 FEED
      AND     Y87  ; LEFT    VAC.CR87
      OR      M220  ; LEFT  Q-RELEASE
      ANI     M304
      ANI     Y63  ; RY STEP0
      OUT     M220  ; LEFT  Q-RELEASE
2444  LD      M220  ; LEFT  Q-RELEASE
      OUT     Y9E  ; LEFT  Q-RELEASE
2446  LD      M74  ; HOLDER  1 CYCLE
      AND     M24  ; VAC.OFF
      AND     M79  ; 2 FEED
      AND     Y88  ; RIGHT   VAC.CR88
      OR      M222  ; RIGHT Q-RELEASE
      ANI     M304
      ANI     Y63  ; RY STEP0
      OUT     M222  ; RIGHT Q-RELEASE
2454  LD      M222  ; RIGHT Q-RELEASE
      OUT     Y9F  ; RIGHT Q-RELEASE
2456  LD      SM400  ; Always  ON
      SET     Y0A0
2458  LDI     X0A0
      AND     X0AF
      AND     X0A1
      MC      N0 M500  ; HOST    DATALINK
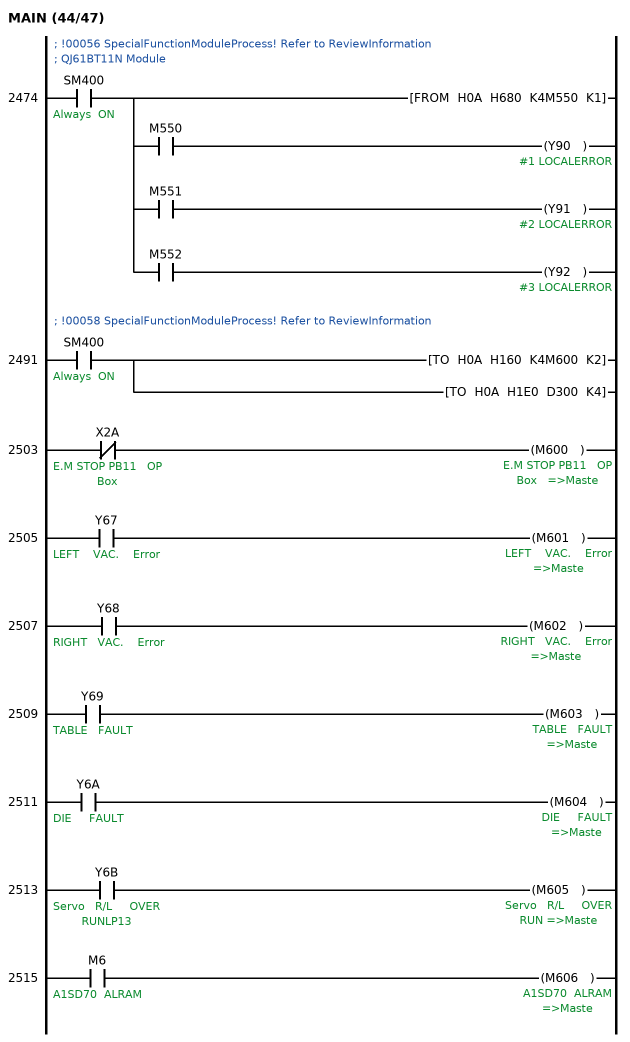
; !00056 SpecialFunctionModuleProcess! Refer to ReviewInformation
; QJ61BT11N Module
2474  LD      SM400  ; Always  ON
      FROM    H0A H680 K4M550 K1
      MPS
      AND     M550
      OUT     Y90  ; #1 LOCALERROR
      MRD
      AND     M551
      OUT     Y91  ; #2 LOCALERROR
      MPP
      AND     M552
      OUT     Y92  ; #3 LOCALERROR
; !00058 SpecialFunctionModuleProcess! Refer to ReviewInformation
2491  LD      SM400  ; Always  ON
      TO      H0A H160 K4M600 K2  ; E.M STOP PB11   OP Box   =>Maste
      TO      H0A H1E0 D300 K4
2503  LDI     X2A  ; E.M STOP PB11   OP Box
      OUT     M600  ; E.M STOP PB11   OP Box   =>Maste
2505  LD      Y67  ; LEFT    VAC.    Error
      OUT     M601  ; LEFT    VAC.    Error    =>Maste
2507  LD      Y68  ; RIGHT   VAC.    Error
      OUT     M602  ; RIGHT   VAC.    Error    =>Maste
2509  LD      Y69  ; TABLE   FAULT
      OUT     M603  ; TABLE   FAULT    =>Maste
2511  LD      Y6A  ; DIE     FAULT
      OUT     M604  ; DIE     FAULT    =>Maste
2513  LD      Y6B  ; Servo   R/L     OVER RUNLP13
      OUT     M605  ; Servo   R/L     OVER RUN =>Maste
2515  LD      M6  ; A1SD70  ALRAM
      OUT     M606  ; A1SD70  ALRAM    =>Maste
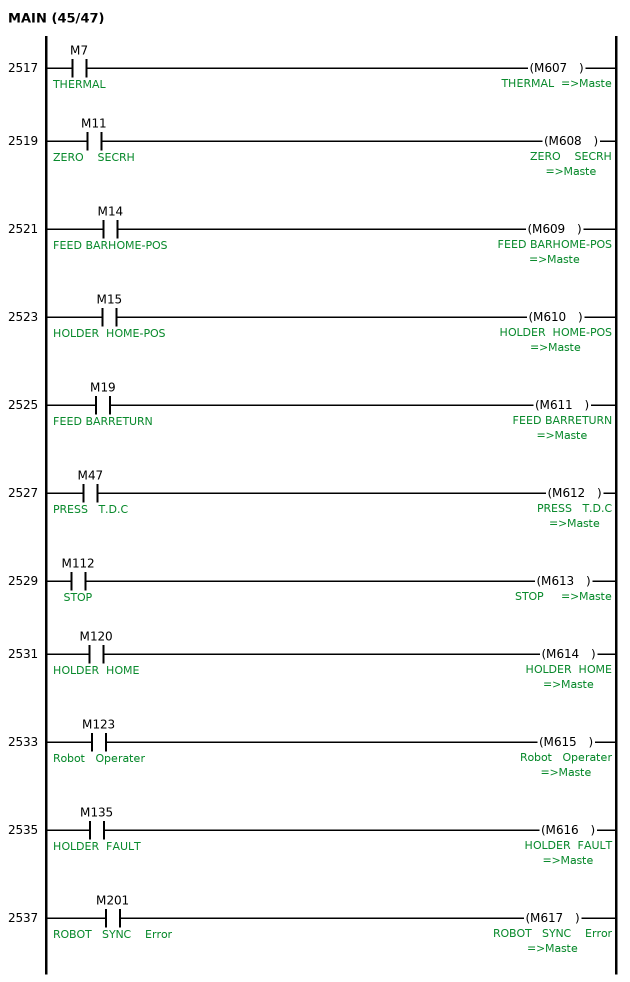
2517  LD      M7  ; THERMAL
      OUT     M607  ; THERMAL  =>Maste
2519  LD      M11  ; ZERO    SECRH
      OUT     M608  ; ZERO    SECRH    =>Maste
2521  LD      M14  ; FEED BARHOME-POS
      OUT     M609  ; FEED BARHOME-POS =>Maste
2523  LD      M15  ; HOLDER  HOME-POS
      OUT     M610  ; HOLDER  HOME-POS =>Maste
2525  LD      M19  ; FEED BARRETURN
      OUT     M611  ; FEED BARRETURN   =>Maste
2527  LD      M47  ; PRESS   T.D.C
      OUT     M612  ; PRESS   T.D.C    =>Maste
2529  LD      M112  ; STOP
      OUT     M613  ; STOP     =>Maste
2531  LD      M120  ; HOLDER  HOME
      OUT     M614  ; HOLDER  HOME     =>Maste
2533  LD      M123  ; Robot   Operater
      OUT     M615  ; Robot   Operater =>Maste
2535  LD      M135  ; HOLDER  FAULT
      OUT     M616  ; HOLDER  FAULT    =>Maste
2537  LD      M201  ; ROBOT   SYNC    Error
      OUT     M617  ; ROBOT   SYNC    Error    =>Maste
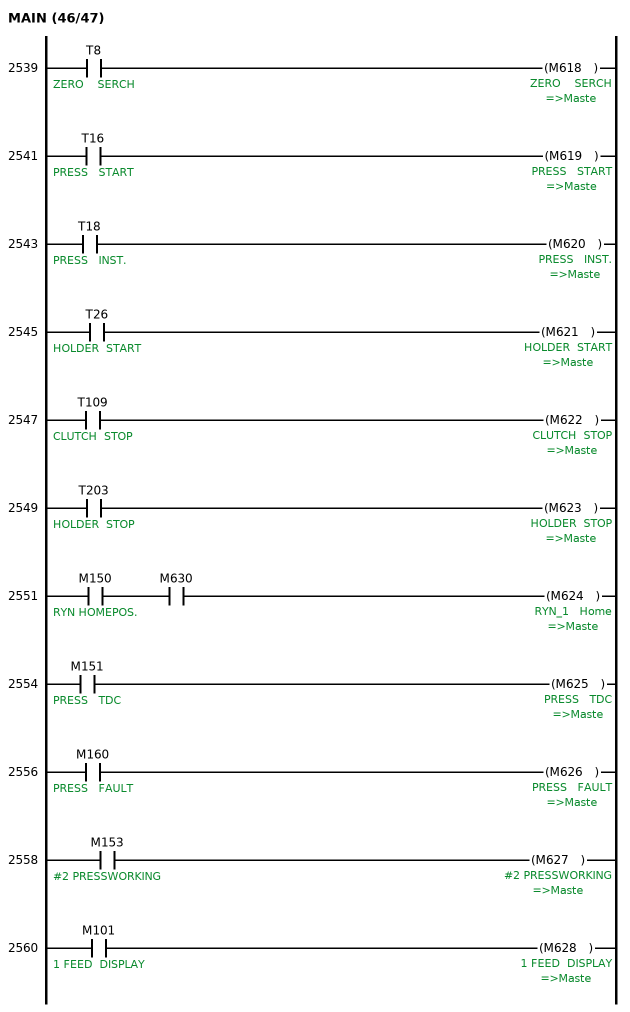
2539  LD      T8  ; ZERO    SERCH
      OUT     M618  ; ZERO    SERCH    =>Maste
2541  LD      T16  ; PRESS   START
      OUT     M619  ; PRESS   START    =>Maste
2543  LD      T18  ; PRESS   INST.
      OUT     M620  ; PRESS   INST.    =>Maste
2545  LD      T26  ; HOLDER  START
      OUT     M621  ; HOLDER  START    =>Maste
2547  LD      T109  ; CLUTCH  STOP
      OUT     M622  ; CLUTCH  STOP     =>Maste
2549  LD      T203  ; HOLDER  STOP
      OUT     M623  ; HOLDER  STOP     =>Maste
2551  LD      M150  ; RYN HOMEPOS.
      AND     M630
      OUT     M624  ; RYN_1   Home     =>Maste
2554  LD      M151  ; PRESS   TDC
      OUT     M625  ; PRESS   TDC      =>Maste
2556  LD      M160  ; PRESS   FAULT
      OUT     M626  ; PRESS   FAULT    =>Maste
2558  LD      M153  ; #2 PRESSWORKING
      OUT     M627  ; #2 PRESSWORKING  =>Maste
2560  LD      M101  ; 1 FEED  DISPLAY
      OUT     M628  ; 1 FEED  DISPLAY  =>Maste
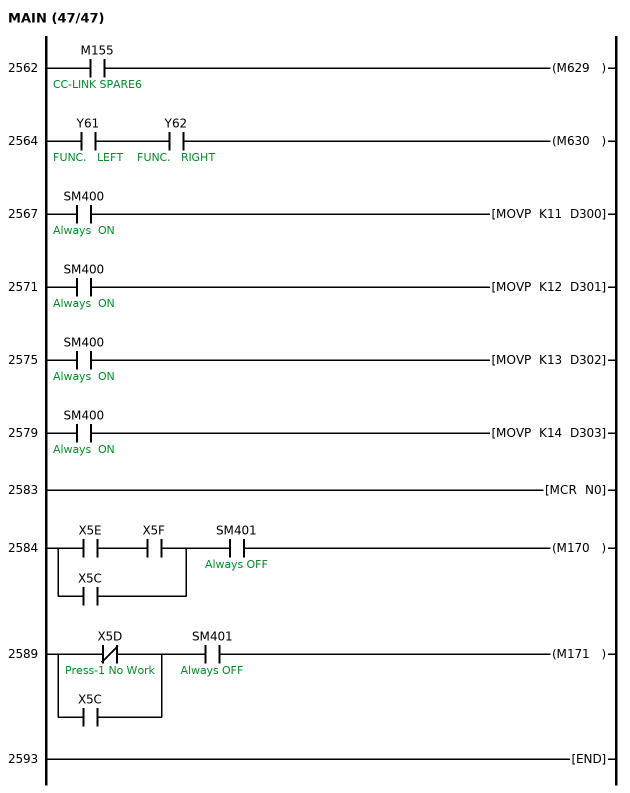
2562  LD      M155  ; CC-LINK SPARE6
      OUT     M629
2564  LD      Y61  ; FUNC.   LEFT
      AND     Y62  ; FUNC.   RIGHT
      OUT     M630
2567  LD      SM400  ; Always  ON
      MOVP    K11 D300
2571  LD      SM400  ; Always  ON
      MOVP    K12 D301
2575  LD      SM400  ; Always  ON
      MOVP    K13 D302
2579  LD      SM400  ; Always  ON
      MOVP    K14 D303
2583  MCR     N0
2584  LD      X5E
      AND     X5F
      OR      X5C
      AND     SM401  ; Always OFF
      OUT     M170
2589  LDI     X5D  ; Press-1 No Work
      OR      X5C
      AND     SM401  ; Always OFF
      OUT     M171
2593  END
END_PROGRAM

// device comments not shown above
X1  ; Synchronization flag
X4  ; Ax#1 M code ON
X5  ; Ax#2 M code ON
X0D  ; Ax#2 BUSY
X11  ; Ax#2 Start completed
X15  ; Ax#2 Positioning completed
X52  ; ¼¾Å¸¸µÈÄÁøÇÑ
X8B  ; ¼¾Å¸¸µÁø°øÀÎÅÍ·Ï
Y0  ; PLC READY
Y5  ; Ax#2 Axis stop
Y0A  ; Ax#2 Forward rotation JOG start
Y0B  ; Ax#2 Reverse rotation JOG start
Y11  ; Axis #2 Positioning start
Y14  ; Ax#1 Execution prohibition flag
Y15  ; Ax#2 Execution prohibition flag
Y8F  ; STEP1COMP.
